SUBAPPLICATION Uebung_175 (* Exercise for E_TABLE_CTRL *)
  (* Standard: 61499-2; Description: Copyright (c) 2023 Meisterschulen am Ostbahnhof This program and the accompanying materials are made available under the terms of the Eclipse Public License 2.0 which is available at https://www.eclipse.org/legal/epl-2.0/ SPDX-License-Identifier: EPL-2.0 *)
  (* Version 1.0, 2025-02-01, Franz Höpfinger, Meisterschulen am Ostbahnhof, initial API and implementation and/or initial documentation *)
  PACKAGE Uebungen;
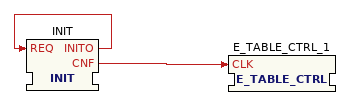
  (* TODO *)
  FBS
    E_TABLE_CTRL_1 : iec61499::events::E_TABLE_CTRL;
    INIT : iec61131::booleanOperators::INIT;
  END_FBS
  EVENT_CONNECTIONS
    INIT.INITO TO INIT.REQ;
    INIT.CNF TO E_TABLE_CTRL_1.CLK;
  END_CONNECTIONS
END_SUBAPPLICATION
